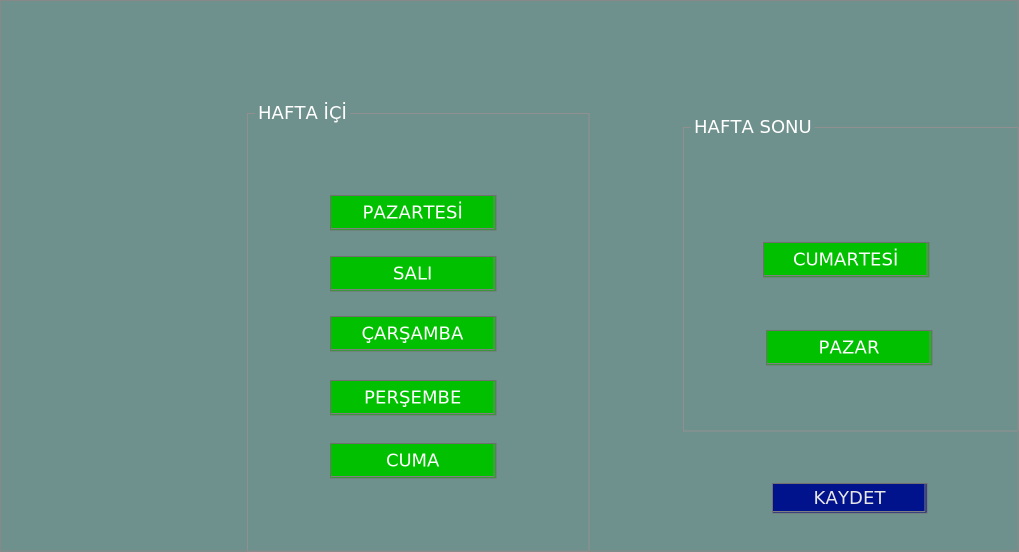
VISUALIZATION mesaiGun_Sayfa  // 1019x552
    GroupBox (247,105 342x447), "HAFTA İÇİ"
        Button (83,90 166x35), "PAZARTESİ", colour toggle: GVL_mesai_gun.pazartesi
            toggle GVL_mesai_gun.pazartesi
        Button (83,151 166x35), "SALI", colour toggle: GVL_mesai_gun.sali
            toggle GVL_mesai_gun.sali
        Button (83,211 166x35), "ÇARŞAMBA", colour toggle: GVL_mesai_gun.carsamba
            toggle GVL_mesai_gun.carsamba
        Button (83,275 166x35), "PERŞEMBE", colour toggle: GVL_mesai_gun.persembe
            toggle GVL_mesai_gun.persembe
        Button (83,338 166x35), "CUMA", colour toggle: GVL_mesai_gun.cuma
            toggle GVL_mesai_gun.cuma
    GroupBox (683,119 336x312), "HAFTA SONU"
        Button (80,123 166x35), "CUMARTESİ", colour toggle: GVL_mesai_gun.cumartesi
            toggle GVL_mesai_gun.cumartesi
        Button (83,211 166x35), "PAZAR", colour toggle: GVL_mesai_gun.pazar
            toggle GVL_mesai_gun.pazar
    Button (772,483 155x30), "KAYDET"
        OnMouseClick: change screen: MesaiSaat_sayfa
END_VISUALIZATION

(* stored: Version 1.1.0.1, ProductVersion 3.1.4024.12
   Visu mesaiGun_Sayfa: Id {96817595-e7bc-48cd-aab4-c1be33147e9d} *)
